// TwinCAT 3 PLC project GarageNCAxis
// ProgramVersion: 3.1.4024.0
// libraries:
//   CmpBitmapPool, * (System)
//   Tc2_MC2, * (Beckhoff Automation GmbH)
//   Tc2_NC, * (Beckhoff Automation GmbH)
//   Tc2_Standard, * (Beckhoff Automation GmbH)
//   Tc2_System, * (Beckhoff Automation GmbH)
//   Tc3_Module, * (Beckhoff Automation GmbH)
// project tree:
//   / GlobalTextList.TcGTLO, PlcTask.TcTTO, Visualization Manager.TcVMO (not stored), VISU_TASK.TcTTO (not stored)
//   POUs/ Blinker.TcPOU (not stored), GarageDoor.TcPOU, ImagePool.TcIPO (not stored), MAIN.TcPOU (not stored), MoveGarageDoor.TcPOU, Visualization.TcVIS
// real-time tasks:
//   TASK PlcTask: cycle T#10ms, priority 20, ADS port 350
//   TASK VISU_TASK: cycle T#200000us, priority 30, ADS port 351
// motion (NC):
//   TASK NC-Task 1 SAF: cycle T#2ms, priority 4, ADS port 501
//   TASK NC-Task 1 SVB: cycle T#10ms, priority 8, ADS port 511
//   AXIS DoorActuator (id 1)
//     OtherSettings: AllowMotionCmdToSlave=true
//     encoder EncType=1
//     drive DrvType=5
//       Analog: TorqueSetpointScale=10, ScaleFactorActTorque=0.1
//       TimeComp: TaskDelayCycles=1
//     controller CtrType=1
//       CtrPara: PriorControlFactor=1
//         Observer: BandWidth=20
// I/O:
//   DEVICE Device 3 (EtherCAT) (disabled), AmsNetId 10.0.30.150.4.1
//     Term 1 (EK1100) [EK1100 EtherCAT Coupler (2A E-Bus)]
//       Term 2 (EL1014) [EL1014 4Ch. Dig. Input 24V, 10µs]
//       Term 3 (EL9011) [EL9011 End Terminal]
// variable links:
//   GarageNCAxis/GarageNCAxis Instance <-> Device 3 (EtherCAT)/Term 1 (EK1100)/Term 2 (EL1014)
//     PlcTask Inputs/GarageDoor.bActuationButton <-> Channel 1/Input
//     PlcTask Inputs/GarageDoor.bErrorButton <-> Channel 2/Input
//   GarageNCAxis/GarageNCAxis Instance <-> NC-Task 1 SAF/Axes/DoorActuator
//     PlcTask Inputs/GarageDoor.fbMotion.Actuator.NcToPlc <-> Outputs/ToPlc
//     PlcTask Outputs/GarageDoor.fbMotion.Actuator.PlcToNc <-> Inputs/FromPlc

CONFIGURATION GarageNCAxis
    RESOURCE PLC ON TwinCAT3
        TASK PlcTask(INTERVAL := T#10ms, PRIORITY := 20);
        PROGRAM MAIN WITH PlcTask : MAIN;
    END_RESOURCE
END_CONFIGURATION

// ---- POUs/GarageDoor.TcPOU
PROGRAM GarageDoor
VAR
	fbMotion : MoveGarageDoor;
	bActuationButton AT %I* : BOOL; //button that we control through visualization
	bErrorButton AT %I* : BOOL; //button for simulating error
	bDoorOpened : BOOL; //sensor for open door
	bDoorClosed : BOOL; //sensor for close door
	bDoorDriveOverload : BOOL; //sensor for the overload of the door
	bDoorPaused : BOOL; //sensor for pausing the door
	bMotionLight : BOOL; //light that indicates there is motion
	fPosition : LREAL; //shows the position of the door
	
	bTest1 : BOOL;
	bTest2 : BOOL;
	bTest3 : BOOL;
	
	bTest4 : BOOL;
	bTest5 : BOOL;
	
	bPauseVis : BOOL;
	bErrorVis : BOOL;

END_VAR

fbMotion.bActuationProgram := bActuationButton;
fbMotion.bError := bErrorButton;

bDoorOpened := fbMotion.bOpened;
bDoorClosed := fbMotion.bClosed;
bDoorDriveOverload := fbMotion.bDriveOverload;
bDoorPaused := fbMotion.bPaused;
bMotionLight := fbMotion.bLight;

fPosition := fbMotion.fActPos;

bTest1 := fbMotion.bVis1O;
bTest2 := fbMotion.bVis2O;
bTest3 := fbMotion.bVis3O;

bTest4 := fbMotion.bVis1C;
bTest5 := fbMotion.bVis2C;

bPauseVis := fbMotion.bPauseImg;
bErrorVis := fbMotion.bErrorImg;


fbMotion();

END_PROGRAM

// ---- POUs/MoveGarageDoor.TcPOU
FUNCTION_BLOCK MoveGarageDoor
VAR_INPUT
	bActuationProgram : BOOL; //actuation button for moving the door
	bError : BOOL; //input error
END_VAR
VAR_OUTPUT
	bClosed : BOOL; //sensor that indicates whether or not the door is closed
	bOpened : BOOL; //sensor that indicates whether or not the door is opened
	bDriveOverload : BOOL; //sensor that indicates whether or not there is an error
	bPaused : BOOL; //sensor that indicates that the door is paused
	bLight : BOOL; //light that shows there is motion
	fActPos : LREAL; //actual position of the axis
	
	bVis1O : BOOL;
	bVis2O : BOOL;
	bVis3O : BOOL;
	bVis1C : BOOL;
	bVis2C : BOOL;
	bErrorImg : BOOL;
	bPauseImg : BOOL;

END_VAR
VAR
	bInitialActivate : BOOL; //helps set the door to closed at the start
	
	fbActivate : R_TRIG;
	fbInitial : R_TRIG; //helps set the initial value to closed
	
	bActuation : BOOL; //works with the actuation program inside of the function block
	
	iState : UDINT;
	
	Actuator : AXIS_REF; //we refrence the axis
	McPower : MC_Power; //power and reset function blocks for the axis
	McReset : MC_Reset;
	McMove : MC_MoveAbsolute;
	McStop : MC_Stop;

	
	bTempC : BOOL; //helps determine what was the door doing before pause/error
	bTempO : BOOL;
	
	fbBlinker : Blinker;
	

END_VAR

bInitialActivate := TRUE; //we close the door at the start
fbInitial(CLK := TRUE);
IF fbInitial.Q THEN
	bClosed := TRUE; //we have set the door to closed at the start (only activates the first time we run the program
END_IF

CASE iState OF
	0:	
		IF McPower.Status THEN
			iState := 10;
		END_IF
	5: //turning actuation off
		bActuation := FALSE;
		iState := 0; //return to the first state
	10:
		fbActivate(CLK := bActuationProgram);
		IF fbActivate.Q THEN
			bActuation := TRUE;
		END_IF
		bTempO := FALSE;
		bTempC := FALSE;
		IF bActuation THEN
			iState := 20; //if we click the button go to the next state and check it's state
		END_IF
	15:
		bActuation := FALSE;
		iState := 100;	
	20:
		IF bClosed THEN
			iState := 40; //open state
		ELSIF bOpened THEN
			iState := 50; //close state
		ELSE
			iState := 999;// driveoverload state
		END_IF
	30:
		bActuation := FALSE;
		iState := 999;
	40: //the door is closed we open it
		bClosed := FALSE;	
		IF bActuation THEN
			bLight := TRUE;
			bTempO := TRUE;
			McMove(Axis := Actuator, //we open the door (100 means openned)
					Position := 1000,
					Velocity := 100,
					Acceleration := 100,
					Deceleration := 100,
					Jerk := 100000,
					Execute := TRUE);
			iState := 45;	
		END_IF
	45:	//check if the movement is done
		fbActivate(CLK := bActuationProgram); //incase we want to pause it
		IF fbActivate.Q THEN
			bActuation := FALSE;
		END_IF
		IF bError THEN
			iState := 30; //incase the door goes to error
		END_IF
		IF bActuation THEN	
			IF McMove.Done AND NOT McMove.Error THEN
				McMove(Axis := Actuator,Execute := FALSE); //we turn it off
				bOpened := TRUE;
				bLight := FALSE;
				iState := 5;
			END_IF
		ELSE
			bPaused := TRUE;
			iState := 15;	
		END_IF
	50: //door is opened we close it
		bOpened := FALSE;	
		IF bActuation THEN
			bLight := TRUE;
			bTempC := TRUE;
			McMove(Axis := Actuator, //we close the door  (0 means openned)
					Position := 0,
					Velocity := 100,
					Acceleration := 100,
					Deceleration := 100,
					Jerk := 100000,
					Execute := TRUE);
			iState := 55; //check if the movement is done
		END_IF	
	55: //check if the movement is done
		fbActivate(CLK := bActuationProgram); //incase we want to pause it
		IF fbActivate.Q THEN
			bActuation := FALSE;
		END_IF
		IF bError THEN
			iState := 30; //incase the door goes to error
		END_IF
		IF bActuation THEN
			
	
			IF McMove.Done AND NOT McMove.Error THEN
				McMove(Axis := Actuator,Execute := FALSE); //we turn it off
				bClosed := TRUE;
				bLight := FALSE;
				iState := 5;
			END_IF
		ELSE
			bPaused := TRUE;
			iState := 15;	
		END_IF
		
	100: //pause state
		//bVis1O := FALSE;
		//bVis2O := FALSE;
		//bVis3O := FALSE;
		//bVis1C := FALSE;
		//bVis2C := FALSE;
		//bPauseImg := TRUE;
		
		bLight := FALSE;
		fbActivate(CLK := bActuationProgram);		
		IF fbActivate.Q THEN
			bActuation := TRUE;
			bPaused := FALSE; //we turn off the pause light
		END_IF
		McStop(Axis := Actuator,
				Deceleration := 300,
				Execute := TRUE);
		IF bActuation AND bTempC THEN
			bLight := TRUE;
			bTempC := FALSE;
			McStop(Axis := Actuator,Execute := FALSE);
			McMove(Axis := Actuator,Execute := FALSE);
			iState := 40;
		ELSIF bActuation AND bTempO THEN
			bLight := TRUE;
			bTempO := FALSE;
			McStop(Axis := Actuator,Execute := FALSE);
			McMove(Axis := Actuator,Execute := FALSE);
			iState := 50;	
		END_IF
				


	999: //error state	
		bErrorImg := TRUE;
		
		bLight := fbBlinker.bBlink;
		fbBlinker();
		bDriveOverload := TRUE;
		fbActivate(CLK := bActuationProgram);		
		IF fbActivate.Q THEN
			bActuation := TRUE;
			bPaused := FALSE; //we turn off the pause light
		END_IF
		McStop(Axis := Actuator,
				Deceleration := 300,
				Execute := TRUE);
		IF bActuation AND bTempC THEN
			bErrorImg := FALSE;
			bDriveOverload := FALSE;
			bLight := TRUE;
			bTempC := FALSE;
			McStop(Axis := Actuator,Execute := FALSE);
			McMove(Axis := Actuator,Execute := FALSE);
			iState := 40;
		ELSIF bActuation AND bTempO THEN
			bErrorImg := FALSE;
			bDriveOverload := FALSE;
			bLight := TRUE;
			bTempO := FALSE;
			McStop(Axis := Actuator,Execute := FALSE);
			McMove(Axis := Actuator,Execute := FALSE);
			iState := 50;	
		END_IF
		
END_CASE
Actuator.ReadStatus(); //referencing the axis to the function blocks
McPower(Axis := Actuator,Enable := TRUE,Enable_Positive := TRUE,Enable_Negative := TRUE);
McReset(Axis := Actuator);
McMove(Axis := Actuator);
McStop(Axis := Actuator);

fActPos := Actuator.NcToPlc.ActPos;

IF bTempO THEN
	//bErrorImg := FALSE;
	//bPauseImg := FALSE;
	bVis1C := FALSE;
	bVis2C := FALSE;
	IF fActPos > 180.0 THEN
		bVis1O := TRUE;
	END_IF
	IF fActPos > 550.0 THEN
		bVis2O := TRUE;
		bVis1O := FALSE;
	END_IF
	IF fActPos > 850.0 THEN
		bVis2O := FALSE;
		bVis3O := TRUE;
	END_IF
END_IF

IF bTempC THEN
	//bErrorImg := FALSE;
	//bPauseImg := FALSE;
	bVis1O := FALSE;
	bVis2O := FALSE;
	IF fActPos < 850.0 THEN
		bVis1C := TRUE;
		bVis3O := FALSE;
	END_IF
	IF fActPos < 550.0 THEN
		bVis2C := TRUE;
		bVis1C := FALSE;
	END_IF
	IF fActPos < 180.0 THEN
		bVis2C := FALSE;
	END_IF
END_IF

END_FUNCTION_BLOCK

// ---- GlobalTextList.TcGTLO
TEXTLIST GlobalTextList
  596 = 'Actuation'
  448 = 'Actuator position'
  961 = 'Closed'
  917 = 'Drive Overload'
  5 = 'Opened'
  837 = 'Paused'
  345 = 'Simulate Error'
END_TEXTLIST

// ---- POUs/Visualization.TcVIS
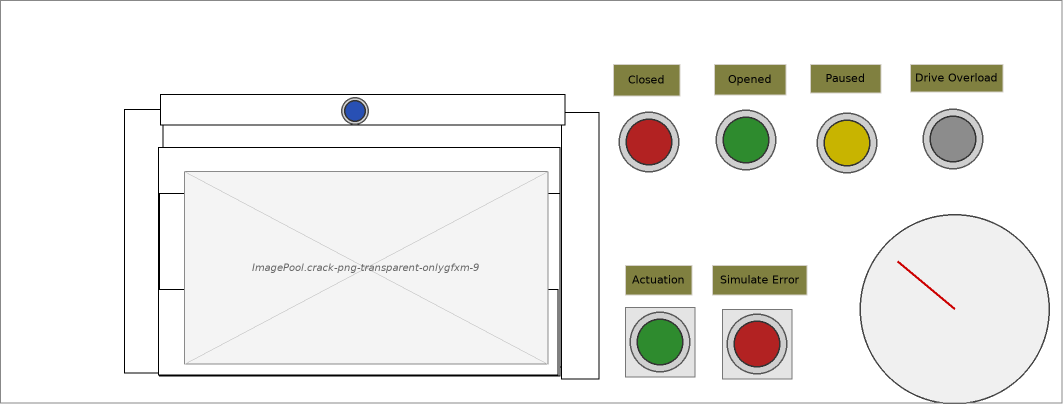
VISUALIZATION Visualization  // 1063x404
    Rectangle (161,123 402x244)
    Rectangle (124,109 39x264)
    Rectangle (561,112 38x267)
    Rectangle (160,94 405x31)
    Lamp1 (339,92 32x38), variable: GarageDoor.bMotionLight, style: Lamp-Lamp1-Blue
    Lamp1 (614,107 70x70), variable: GarageDoor.bDoorClosed, style: Lamp-Lamp1-Red
    Lamp1 (711,105 70x70), variable: GarageDoor.bDoorOpened, style: Lamp-Lamp1-Green
    Lamp1 (812,108 70x70), variable: GarageDoor.bDoorPaused, style: Lamp-Lamp1-Yellow
    Lamp1 (918,104 70x70), variable: GarageDoor.bDoorDriveOverload, style: Lamp-Lamp1-Gray
    PushSwitch (625,307 70x70), variable: GarageDoor.bActuationButton, behaviour: TAP, style: Switch-PushSwitch-Green
    PushSwitch (722,309 70x70), variable: GarageDoor.bErrorButton, behaviour: TAP, style: Switch-PushSwitch-Red
    Rectangle (161,274 399x96), invisible if: NOT GarageDoor.bTest1
    Rectangle (158,147 402x225), invisible if: NOT GarageDoor.bTest3
    Rectangle (160,205 399x166), invisible if: NOT GarageDoor.bTest2
    Rectangle (159,193 401x183), invisible if: NOT GarageDoor.bTest4
    Rectangle (158,289 400x86), invisible if: NOT GarageDoor.bTest5
    Image (184,171 364x193), invisible if: NOT GarageDoor.bErrorVis, image: ImagePool.crack-png-transparent-onlygfxm-9
    Meter360 (846,214 217x190), value: GarageDoor.fPosition, style: Meter-Meter360-Gray, scale format: %.1f, scale 0..1000
        p518627256: Actuator position
    Textfield (613,64 67x32), "Closed", colour toggle: GarageDoor.bDoorClosed
    Textfield (714,64 72x31), "Opened", colour toggle: GarageDoor.bDoorOpened
    Textfield (810,64 71x29), "Paused", colour toggle: GarageDoor.bDoorPaused
    Textfield (910,64 93x28), "Drive Overload", colour toggle: GarageDoor.bDoorDriveOverload
    Textfield (625,265 67x30), "Actuation", colour toggle: GarageDoor.bActuationButton
    Textfield (712,265 95x30), "Simulate Error", colour toggle: GarageDoor.bErrorButton
END_VISUALIZATION
